TYPE ST_EL3022 :
STRUCT
	
	//2-channel analog input
	rPressureRegulator	:	LREAL; //Terminal 17 SMC low differential pressure sensor
	
END_STRUCT
END_TYPE

(* stored: Version 1.1.0.1, ProductVersion 3.1.4024.12
   DUT ST_EL3022: Id {d3b0cf3d-d3b0-4137-ace9-ed3ec36236fd} *)
